// TIA Portal V18 export
VAR_GLOBAL   // PLC tag table "05 Tracking"
END_VAR
VAR_GLOBAL CONSTANT   // user constants
   tracking_N_pezzi : Int := 10;
   NumCharTrackingArticle : Int := 30;
   NumCharTrackingId : Int := 30;
   NumCharTrackingLotto : Int := 30;
   NumCharTrackingProfile : Int := 30;
   NumCharTrackingStazione : Int := 30;
   tr01_BSL : Int := 1;
   tr02_Rull1_Acc : Int := 2;
   tr03_Rull2_Rastr : Int := 3;
   tr04_Rull3_Prel : Int := 4;
   tr05_Robot : Int := 5;
   tr06_deposito : Int := 6;
END_VAR
